{attribute 'GeneratedUsingTerminal: KL6211'}
{attribute addProperty BoxType "KL6211"}
{attribute addProperty Description ""}
{attribute addProperty Physics ""}
{attribute addProperty Id "Channel_1AT %Q*Channel_879058310"}
{attribute addProperty CRC "1611886241"}
{attribute addProperty Size "0"}
TYPE KL6211_60136EA1 :
STRUCT
	{attribute addProperty Name "Channel_1"}
	Channel_1 : Channel_87905831;
END_STRUCT
END_TYPE

(* stored: Version 1.2.0.0, ProductVersion 3.1.4024.9
   DUT KL6211_60136EA1: Id {949c1962-57ac-441b-aaa7-8cb76b437f22} *)
